(* Logix 5000 project; controller DUNEW2PLC1 vendor 1 type 14 code 221 rev 33.11; software revision 33.00; part 5 of 7 *)
(* tags used below, declared in another part *)
   AbortQueue : BOOL;
   ALL_EOT_GOOD : BOOL;
   btm_support_collision_ymax : DINT;
   btm_support_collision_ymin : DINT;
   ERROR_CODE : DINT;
   FRAME_LOC_FT_BTM : BOOL;
   FRAME_LOC_FT_MID : BOOL;
   FRAME_LOC_FT_TOP : BOOL;
   FRAME_LOC_HD_BTM : BOOL;
   FRAME_LOC_HD_MID : BOOL;
   FRAME_LOC_HD_TOP : BOOL;
   INIT_DONE : BOOL;
   mid_support_collision_ymax : DINT;
   mid_support_collision_ymin : DINT;
   MINUS_X_EOT : BOOL;
   MINUS_Y_EOT : BOOL;
   MOVE_TYPE : INT;   // 0 = No Move 1 = XY JOG 2 = XY Plane Move 3 = Z JOG 4 = Z Axis Move 5 = Toggle Latch Actuator 6 = Home the Latch Actuator
   NEXTSTATE : DINT;
   PLUS_X_EOT : BOOL;
   PLUS_Y_EOT : BOOL;
   STATE : DINT;   // CURRENT State Machine State
   STATE_REQUEST : DINT;
   top_support_collision_ymax : DINT;
   top_support_collision_ymin : DINT;
   X_axis : AXIS_CIP_DRIVE;
   X_XFER_OK : BOOL;   // If at the head, check head support arms. Same for foot
   X_Y : COORDINATE_SYSTEM;
   xz : COORDINATE_SYSTEM;
   xz_position_target : REAL[2];
   xz_speed : DINT;
   Y_axis : AXIS_CIP_DRIVE;
   Y_XFER_OK : BOOL;
   yz : COORDINATE_SYSTEM;
   yz_position_target : REAL[2];
   yz_speed : DINT;
   Z_axis : AXIS_CIP_DRIVE;
   Z_EOT : BOOL;
   Z_RETRACTED : BOOL;

PROGRAM state_10_error   (* main routine main *)
VAR
   error_axes_stopped_ob : BOOL;
   error_axes_stopped_sb : BOOL := 1;
   error_entry_ob : BOOL;
   error_entry_sb : BOOL;
   error_servo_off : BOOL;
   error_servoed_off_ob : BOOL;
   error_servoed_off_sb : BOOL;
   STATE10_IND : BOOL; {access Read Only}
   x_axis_mafr : MOTION_INSTRUCTION := (FLAGS := 33554432);
   x_axis_msf : MOTION_INSTRUCTION := (FLAGS := 33554432);
   xy_error_stop_control : MOTION_INSTRUCTION := (FLAGS := 704643072, DN := 1, PC := 1);
   y_axis_mafr : MOTION_INSTRUCTION := (FLAGS := 33554432);
   y_axis_msf : MOTION_INSTRUCTION := (FLAGS := 33554432);
   z_axis_error_stop_control : MOTION_INSTRUCTION := (FLAGS := 704643072, DN := 1, PC := 1);
   z_axis_mafr : MOTION_INSTRUCTION := (FLAGS := 33554432);
   z_axis_msf : MOTION_INSTRUCTION := (FLAGS := 33554432);
END_VAR

ROUTINE main   (* ladder *)
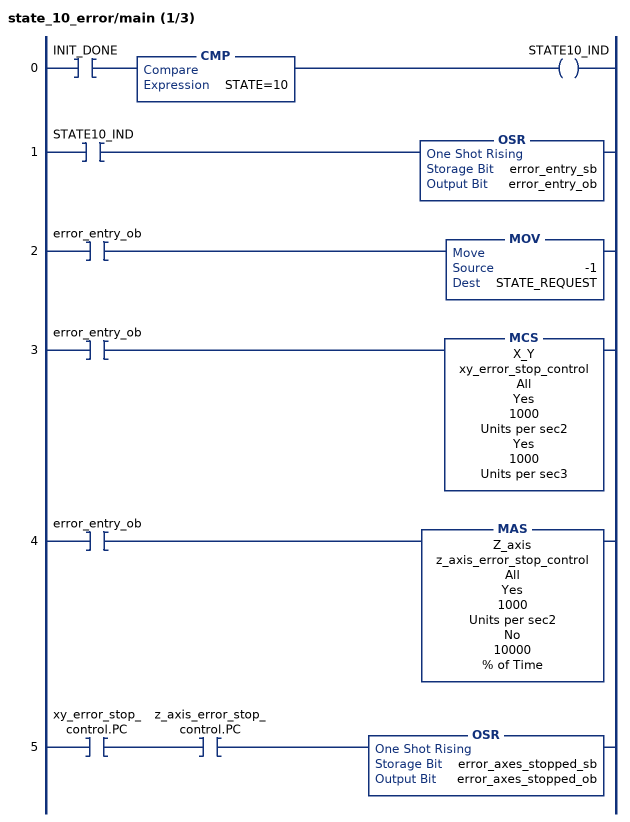
   0: XIC(INIT_DONE)CMP(STATE=10)OTE(STATE10_IND);
   1: XIC(STATE10_IND)OSR(error_entry_sb,error_entry_ob);
   2: XIC(error_entry_ob)MOV(-1,STATE_REQUEST);
   3: XIC(error_entry_ob)MCS(X_Y,xy_error_stop_control,All,Yes,1000,Units per sec2,Yes,1000,Units per sec3);
   4: XIC(error_entry_ob)MAS(Z_axis,z_axis_error_stop_control,All,Yes,1000,Units per sec2,No,10000,% of Time);
   5: XIC(xy_error_stop_control.PC)XIC(z_axis_error_stop_control.PC)OSR(error_axes_stopped_sb,error_axes_stopped_ob);
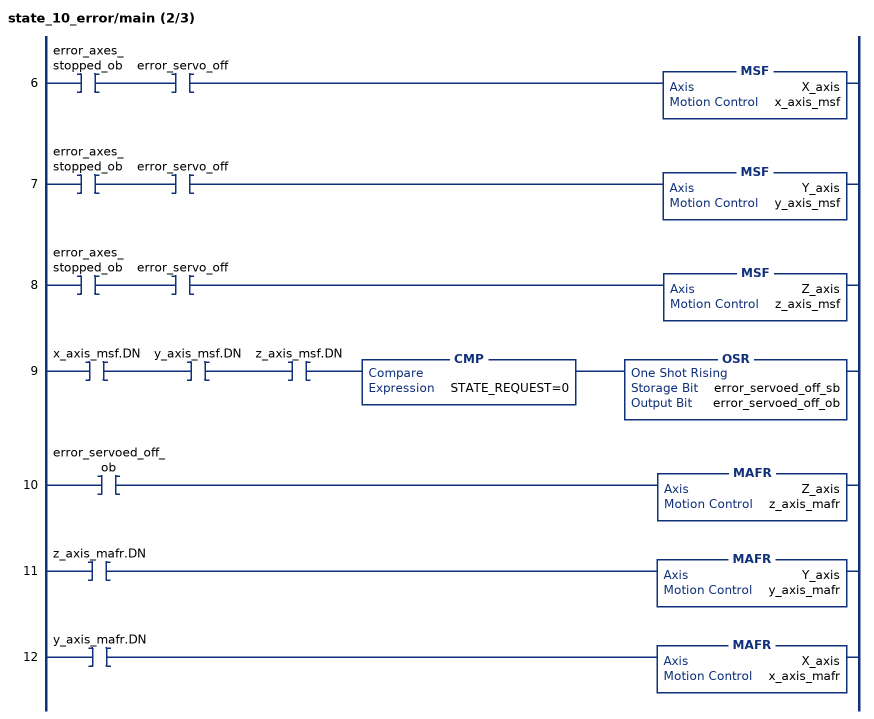
   6: XIC(error_axes_stopped_ob)XIC(error_servo_off)MSF(X_axis,x_axis_msf);
   7: XIC(error_axes_stopped_ob)XIC(error_servo_off)MSF(Y_axis,y_axis_msf);
   8: XIC(error_axes_stopped_ob)XIC(error_servo_off)MSF(Z_axis,z_axis_msf);
   9: XIC(x_axis_msf.DN)XIC(y_axis_msf.DN)XIC(z_axis_msf.DN)CMP(STATE_REQUEST=0)OSR(error_servoed_off_sb,error_servoed_off_ob);
   10: XIC(error_servoed_off_ob)MAFR(Z_axis,z_axis_mafr);
   11: XIC(z_axis_mafr.DN)MAFR(Y_axis,y_axis_mafr);
   12: XIC(y_axis_mafr.DN)MAFR(X_axis,x_axis_mafr);
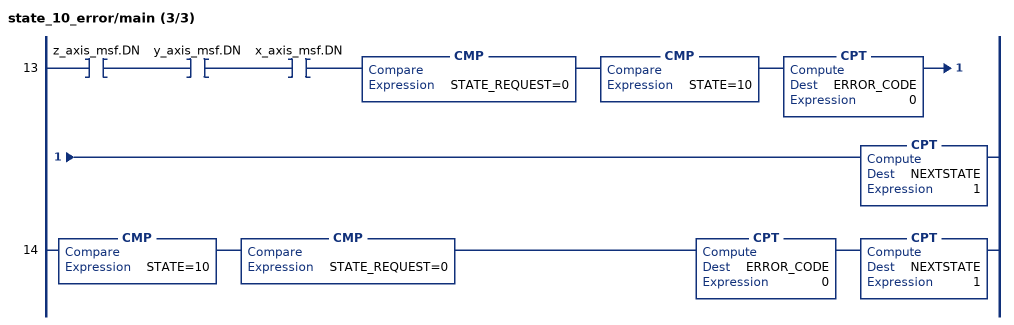
   13: XIC(z_axis_msf.DN)XIC(y_axis_msf.DN)XIC(x_axis_msf.DN)CMP(STATE_REQUEST=0)CMP(STATE=10)CPT(ERROR_CODE,0)CPT(NEXTSTATE,1);
   14: CMP(STATE=10)CMP(STATE_REQUEST=0)CPT(ERROR_CODE,0)CPT(NEXTSTATE,1);
END_ROUTINE
END_PROGRAM

PROGRAM state_11_eot_trip   (* main routine main *)
VAR
   eot_axes_enabled : BOOL := 1;
   eot_entry_ob : BOOL;
   eot_entry_sb : BOOL;
   eot_manual_ob : BOOL;
   eot_manual_sb : BOOL;
   eot_mso_start_ob : BOOL;
   eot_mso_start_sb : BOOL;
   eot_mso_x : MOTION_INSTRUCTION := (FLAGS := 536870912, DN := 1);
   eot_mso_y : MOTION_INSTRUCTION := (FLAGS := 536870912, DN := 1);
   eot_mso_z : MOTION_INSTRUCTION := (FLAGS := 536870912, DN := 1);
   eot_recover_ready : BOOL;
   eot_recovery_done : BOOL;
   eot_stop_x : MOTION_INSTRUCTION := (FLAGS := 671088640, DN := 1, PC := 1);
   eot_stop_xy : MOTION_INSTRUCTION := (FLAGS := 671088640, DN := 1, PC := 1);
   eot_stop_xz : MOTION_INSTRUCTION := (FLAGS := 671088640, DN := 1, PC := 1);
   eot_stop_y : MOTION_INSTRUCTION := (FLAGS := 671088640, DN := 1, PC := 1);
   eot_stop_yz : MOTION_INSTRUCTION := (FLAGS := 704643072, DN := 1, PC := 1);
   eot_stop_z : MOTION_INSTRUCTION := (FLAGS := 671088640, DN := 1, PC := 1);
   eot_stops_done : BOOL;
   STATE11_IND : BOOL; {access Read Only}
   x_minus_clear_ob : BOOL;
   x_minus_clear_sb : BOOL;
   x_minus_cleared : BOOL;
   x_minus_jog_active : BOOL;
   x_minus_jog_cmd : MOTION_INSTRUCTION;
   x_minus_jog_start_ob : BOOL;
   x_minus_jog_start_sb : BOOL;
   x_minus_jog_stop : MOTION_INSTRUCTION;
   x_minus_jog_timer : TIMER := (PRE := 10000);
   x_minus_mrp_cmd : MOTION_INSTRUCTION;
   x_minus_mrp_start_ob : BOOL;
   x_minus_mrp_start_sb : BOOL;
   x_minus_stop_req : BOOL;
   x_minus_timeout : BOOL;
   x_minus_trip : BOOL;
   x_plus_clear_ob : BOOL;
   x_plus_clear_sb : BOOL;
   x_plus_jog_active : BOOL;
   x_plus_jog_cmd : MOTION_INSTRUCTION := (FLAGS := 536870912, DN := 1);
   x_plus_jog_start_ob : BOOL;
   x_plus_jog_start_sb : BOOL;
   x_plus_jog_stop : MOTION_INSTRUCTION := (FLAGS := 671088640, DN := 1, PC := 1);
   x_plus_jog_timer : TIMER := (PRE := 10000);
   x_plus_stop_req : BOOL;
   x_plus_timeout : BOOL;
   x_plus_trip : BOOL;
   y_minus_clear_ob : BOOL;
   y_minus_clear_sb : BOOL;
   y_minus_cleared : BOOL;
   y_minus_jog_active : BOOL;
   y_minus_jog_cmd : MOTION_INSTRUCTION;
   y_minus_jog_start_ob : BOOL;
   y_minus_jog_start_sb : BOOL;
   y_minus_jog_stop : MOTION_INSTRUCTION;
   y_minus_jog_timer : TIMER := (PRE := 10000);
   y_minus_mrp_cmd : MOTION_INSTRUCTION;
   y_minus_mrp_start_ob : BOOL;
   y_minus_mrp_start_sb : BOOL;
   y_minus_stop_req : BOOL;
   y_minus_timeout : BOOL;
   y_minus_trip : BOOL;
   y_plus_clear_ob : BOOL;
   y_plus_clear_sb : BOOL;
   y_plus_jog_active : BOOL;
   y_plus_jog_cmd : MOTION_INSTRUCTION;
   y_plus_jog_start_ob : BOOL;
   y_plus_jog_start_sb : BOOL;
   y_plus_jog_stop : MOTION_INSTRUCTION;
   y_plus_jog_timer : TIMER := (PRE := 10000);
   y_plus_stop_req : BOOL;
   y_plus_timeout : BOOL;
   y_plus_trip : BOOL;
   z_recover_started : BOOL;
   z_trip : BOOL;
   z_zero_cmd : MOTION_INSTRUCTION;
   z_zero_start_ob : BOOL;
   z_zero_start_sb : BOOL;
END_VAR

ROUTINE main   (* ladder *)
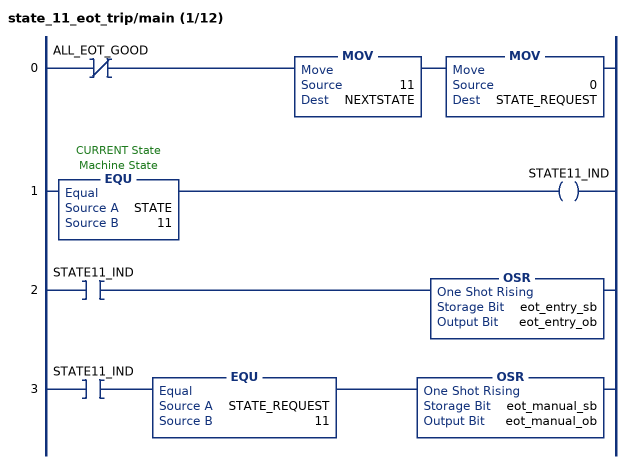
   0: XIO(ALL_EOT_GOOD)MOV(11,NEXTSTATE)MOV(0,STATE_REQUEST);
   1: EQU(STATE,11)OTE(STATE11_IND);
   2: XIC(STATE11_IND)OSR(eot_entry_sb,eot_entry_ob);
   3: XIC(STATE11_IND)EQU(STATE_REQUEST,11)OSR(eot_manual_sb,eot_manual_ob);
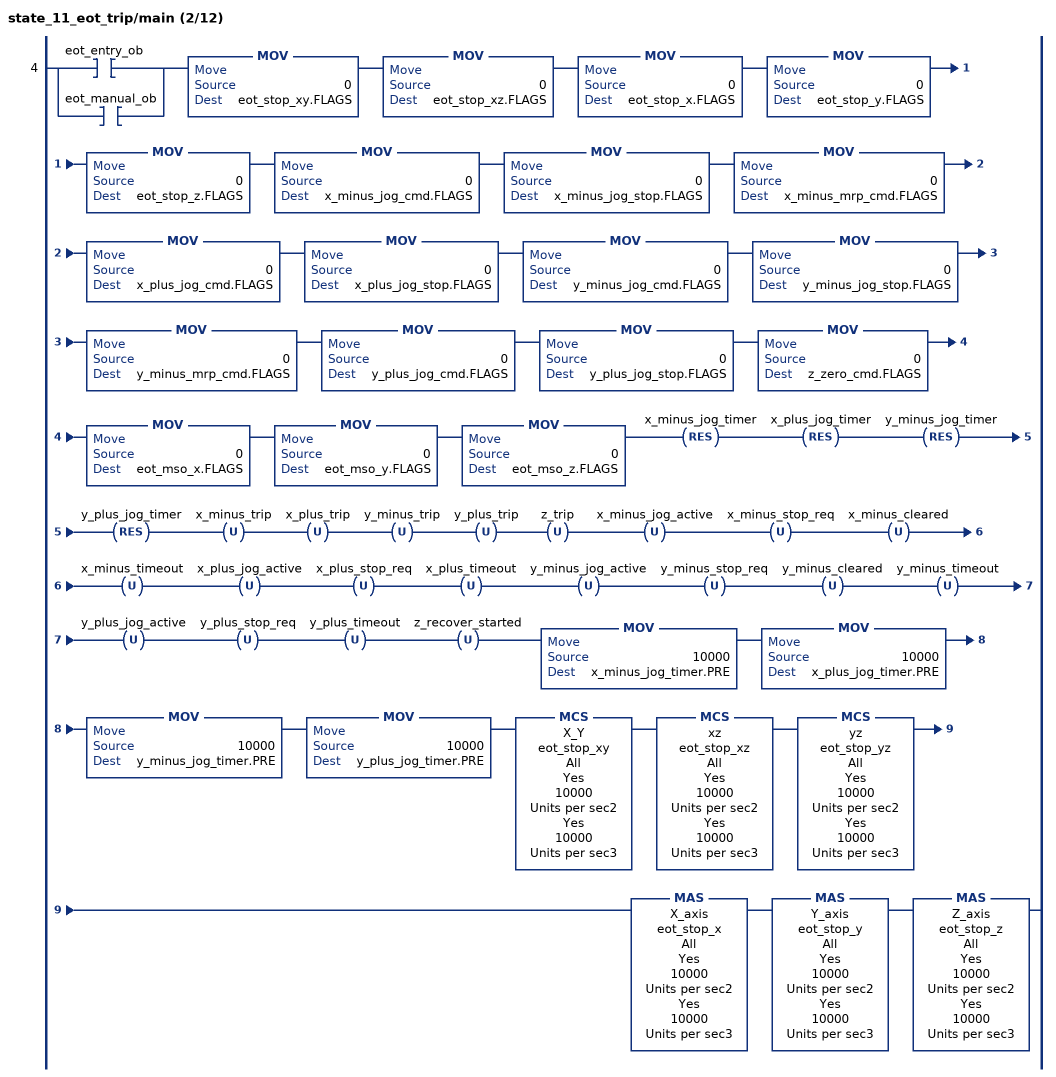
   4: [XIC(eot_entry_ob) ,XIC(eot_manual_ob) ]MOV(0,eot_stop_xy.FLAGS)MOV(0,eot_stop_xz.FLAGS)MOV(0,eot_stop_x.FLAGS)MOV(0,eot_stop_y.FLAGS)MOV(0,eot_stop_z.FLAGS)MOV(0,x_minus_jog_cmd.FLAGS)MOV(0,x_minus_jog_stop.FLAGS)MOV(0,x_minus_mrp_cmd.FLAGS)MOV(0,x_plus_jog_cmd.FLAGS)MOV(0,x_plus_jog_stop.FLAGS)MOV(0,y_minus_jog_cmd.FLAGS)MOV(0,y_minus_jog_stop.FLAGS)MOV(0,y_minus_mrp_cmd.FLAGS)MOV(0,y_plus_jog_cmd.FLAGS)MOV(0,y_plus_jog_stop.FLAGS)MOV(0,z_zero_cmd.FLAGS)MOV(0,eot_mso_x.FLAGS)MOV(0,eot_mso_y.FLAGS)MOV(0,eot_mso_z.FLAGS)RES(x_minus_jog_timer)RES(x_plus_jog_timer)RES(y_minus_jog_timer)RES(y_plus_jog_timer)OTU(x_minus_trip)OTU(x_plus_trip)OTU(y_minus_trip)OTU(y_plus_trip)OTU(z_trip)OTU(x_minus_jog_active)OTU(x_minus_stop_req)OTU(x_minus_cleared)OTU(x_minus_timeout)OTU(x_plus_jog_active)OTU(x_plus_stop_req)OTU(x_plus_timeout)OTU(y_minus_jog_active)OTU(y_minus_stop_req)OTU(y_minus_cleared)OTU(y_minus_timeout)OTU(y_plus_jog_active)OTU(y_plus_stop_req)OTU(y_plus_timeout)OTU(z_recover_started)MOV(10000,x_minus_jog_timer.PRE)MOV(10000,x_plus_jog_timer.PRE)MOV(10000,y_minus_jog_timer.PRE)MOV(10000,y_plus_jog_timer.PRE)MCS(X_Y,eot_stop_xy,All,Yes,10000,Units per sec2,Yes,10000,Units per sec3)MCS(xz,eot_stop_xz,All,Yes,10000,Units per sec2,Yes,10000,Units per sec3)MCS(yz,eot_stop_yz,All,Yes,10000,Units per sec2,Yes,10000,Units per sec3)MAS(X_axis,eot_stop_x,All,Yes,10000,Units per sec2,Yes,10000,Units per sec3)MAS(Y_axis,eot_stop_y,All,Yes,10000,Units per sec2,Yes,10000,Units per sec3)MAS(Z_axis,eot_stop_z,All,Yes,10000,Units per sec2,Yes,10000,Units per sec3);
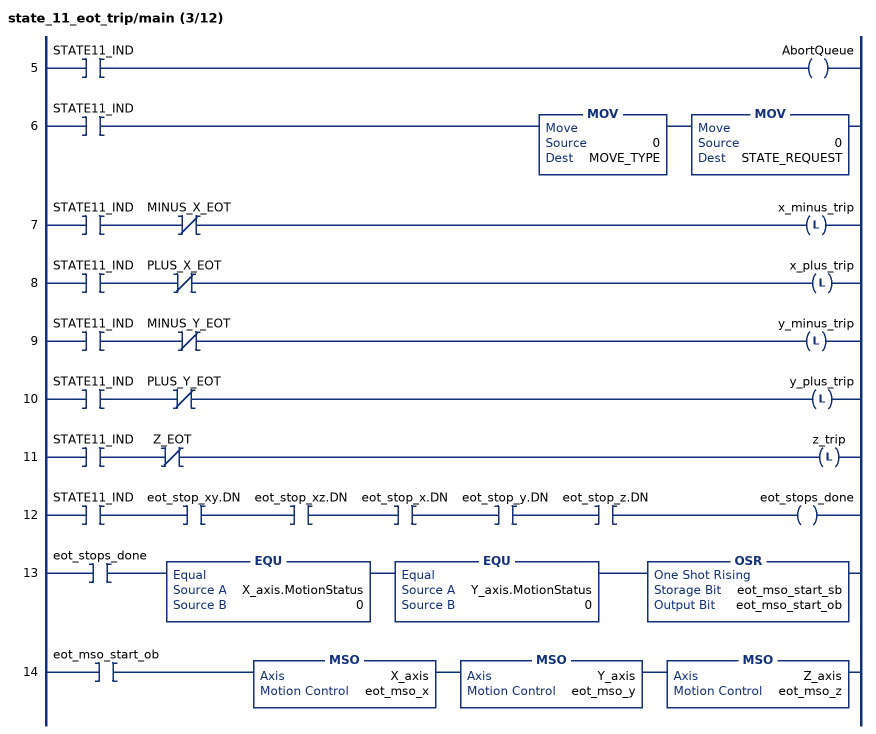
   5: XIC(STATE11_IND)OTE(AbortQueue);
   6: XIC(STATE11_IND)MOV(0,MOVE_TYPE)MOV(0,STATE_REQUEST);
   7: XIC(STATE11_IND)XIO(MINUS_X_EOT)OTL(x_minus_trip);
   8: XIC(STATE11_IND)XIO(PLUS_X_EOT)OTL(x_plus_trip);
   9: XIC(STATE11_IND)XIO(MINUS_Y_EOT)OTL(y_minus_trip);
   10: XIC(STATE11_IND)XIO(PLUS_Y_EOT)OTL(y_plus_trip);
   11: XIC(STATE11_IND)XIO(Z_EOT)OTL(z_trip);
   12: XIC(STATE11_IND)XIC(eot_stop_xy.DN)XIC(eot_stop_xz.DN)XIC(eot_stop_x.DN)XIC(eot_stop_y.DN)XIC(eot_stop_z.DN)OTE(eot_stops_done);
   13: XIC(eot_stops_done)EQU(X_axis.MotionStatus,0)EQU(Y_axis.MotionStatus,0)OSR(eot_mso_start_sb,eot_mso_start_ob);
   14: XIC(eot_mso_start_ob)MSO(X_axis,eot_mso_x)MSO(Y_axis,eot_mso_y)MSO(Z_axis,eot_mso_z);
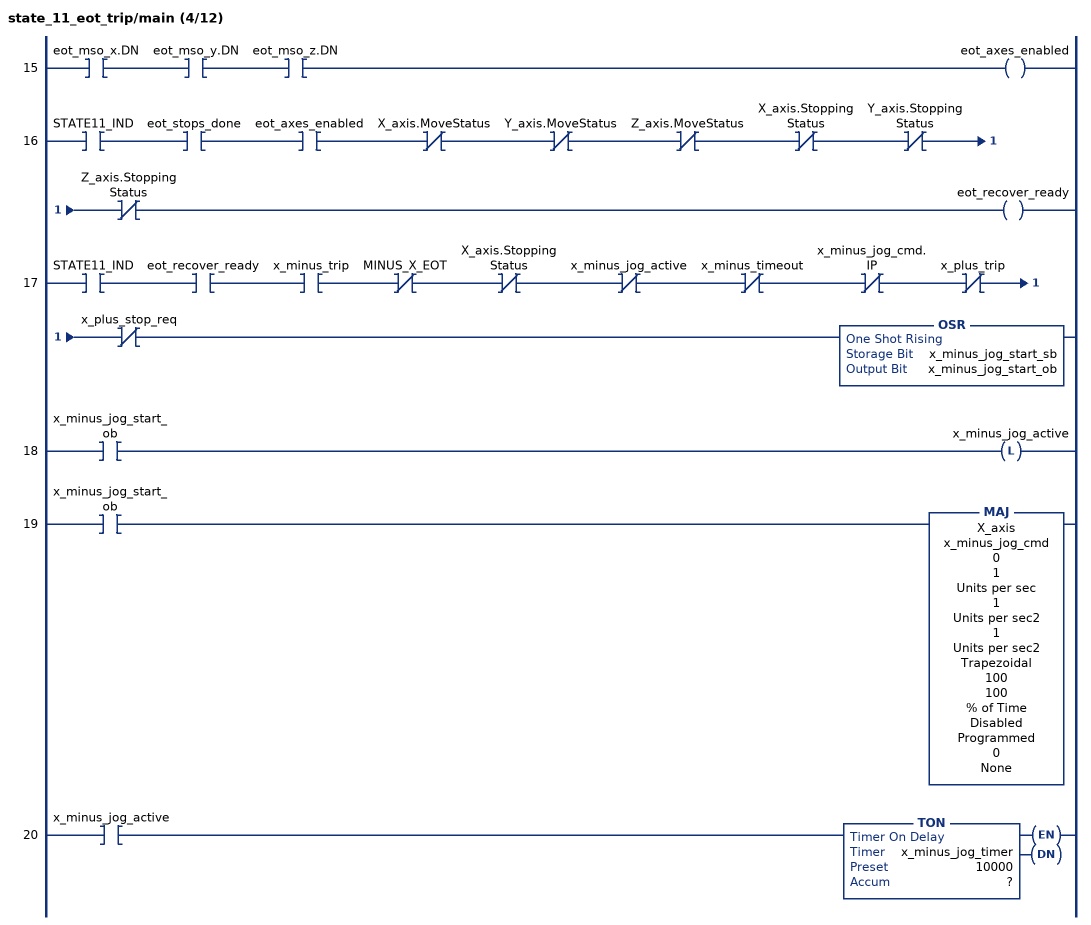
   15: XIC(eot_mso_x.DN)XIC(eot_mso_y.DN)XIC(eot_mso_z.DN)OTE(eot_axes_enabled);
   16: XIC(STATE11_IND)XIC(eot_stops_done)XIC(eot_axes_enabled)XIO(X_axis.MoveStatus)XIO(Y_axis.MoveStatus)XIO(Z_axis.MoveStatus)XIO(X_axis.StoppingStatus)XIO(Y_axis.StoppingStatus)XIO(Z_axis.StoppingStatus)OTE(eot_recover_ready);
   17: XIC(STATE11_IND)XIC(eot_recover_ready)XIC(x_minus_trip)XIO(MINUS_X_EOT)XIO(X_axis.StoppingStatus)XIO(x_minus_jog_active)XIO(x_minus_timeout)XIO(x_minus_jog_cmd.IP)XIO(x_plus_trip)XIO(x_plus_stop_req)OSR(x_minus_jog_start_sb,x_minus_jog_start_ob);
   18: XIC(x_minus_jog_start_ob)OTL(x_minus_jog_active);
   19: XIC(x_minus_jog_start_ob)MAJ(X_axis,x_minus_jog_cmd,0,1,Units per sec,1,Units per sec2,1,Units per sec2,Trapezoidal,100,100,% of Time,Disabled,Programmed,0,None);
   20: XIC(x_minus_jog_active)TON(x_minus_jog_timer,?,?);
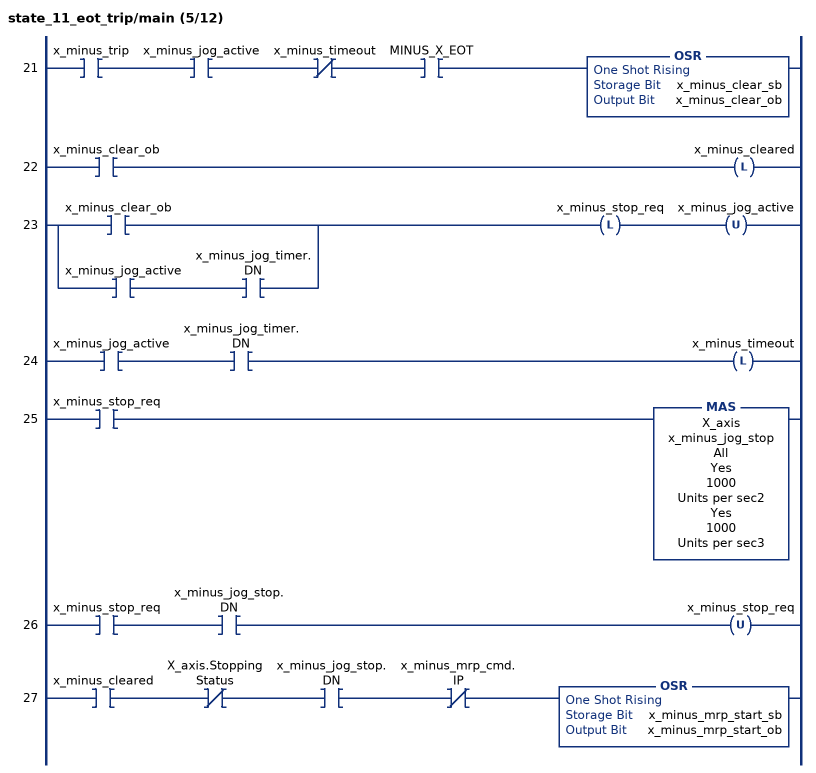
   21: XIC(x_minus_trip)XIC(x_minus_jog_active)XIO(x_minus_timeout)XIC(MINUS_X_EOT)OSR(x_minus_clear_sb,x_minus_clear_ob);
   22: XIC(x_minus_clear_ob)OTL(x_minus_cleared);
   23: [XIC(x_minus_clear_ob) ,XIC(x_minus_jog_active) XIC(x_minus_jog_timer.DN) ]OTL(x_minus_stop_req)OTU(x_minus_jog_active);
   24: XIC(x_minus_jog_active)XIC(x_minus_jog_timer.DN)OTL(x_minus_timeout);
   25: XIC(x_minus_stop_req)MAS(X_axis,x_minus_jog_stop,All,Yes,1000,Units per sec2,Yes,1000,Units per sec3);
   26: XIC(x_minus_stop_req)XIC(x_minus_jog_stop.DN)OTU(x_minus_stop_req);
   27: XIC(x_minus_cleared)XIO(X_axis.StoppingStatus)XIC(x_minus_jog_stop.DN)XIO(x_minus_mrp_cmd.IP)OSR(x_minus_mrp_start_sb,x_minus_mrp_start_ob);
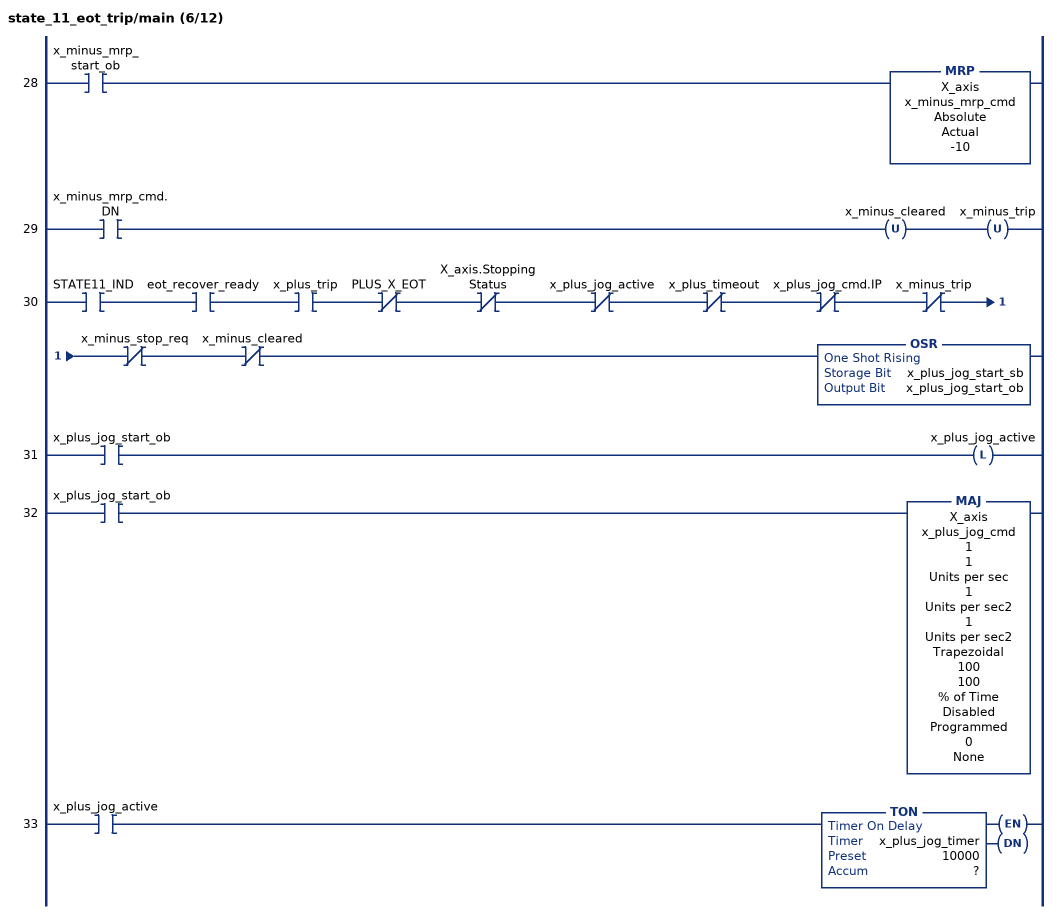
   28: XIC(x_minus_mrp_start_ob)MRP(X_axis,x_minus_mrp_cmd,Absolute,Actual,-10);
   29: XIC(x_minus_mrp_cmd.DN)OTU(x_minus_cleared)OTU(x_minus_trip);
   30: XIC(STATE11_IND)XIC(eot_recover_ready)XIC(x_plus_trip)XIO(PLUS_X_EOT)XIO(X_axis.StoppingStatus)XIO(x_plus_jog_active)XIO(x_plus_timeout)XIO(x_plus_jog_cmd.IP)XIO(x_minus_trip)XIO(x_minus_stop_req)XIO(x_minus_cleared)OSR(x_plus_jog_start_sb,x_plus_jog_start_ob);
   31: XIC(x_plus_jog_start_ob)OTL(x_plus_jog_active);
   32: XIC(x_plus_jog_start_ob)MAJ(X_axis,x_plus_jog_cmd,1,1,Units per sec,1,Units per sec2,1,Units per sec2,Trapezoidal,100,100,% of Time,Disabled,Programmed,0,None);
   33: XIC(x_plus_jog_active)TON(x_plus_jog_timer,?,?);
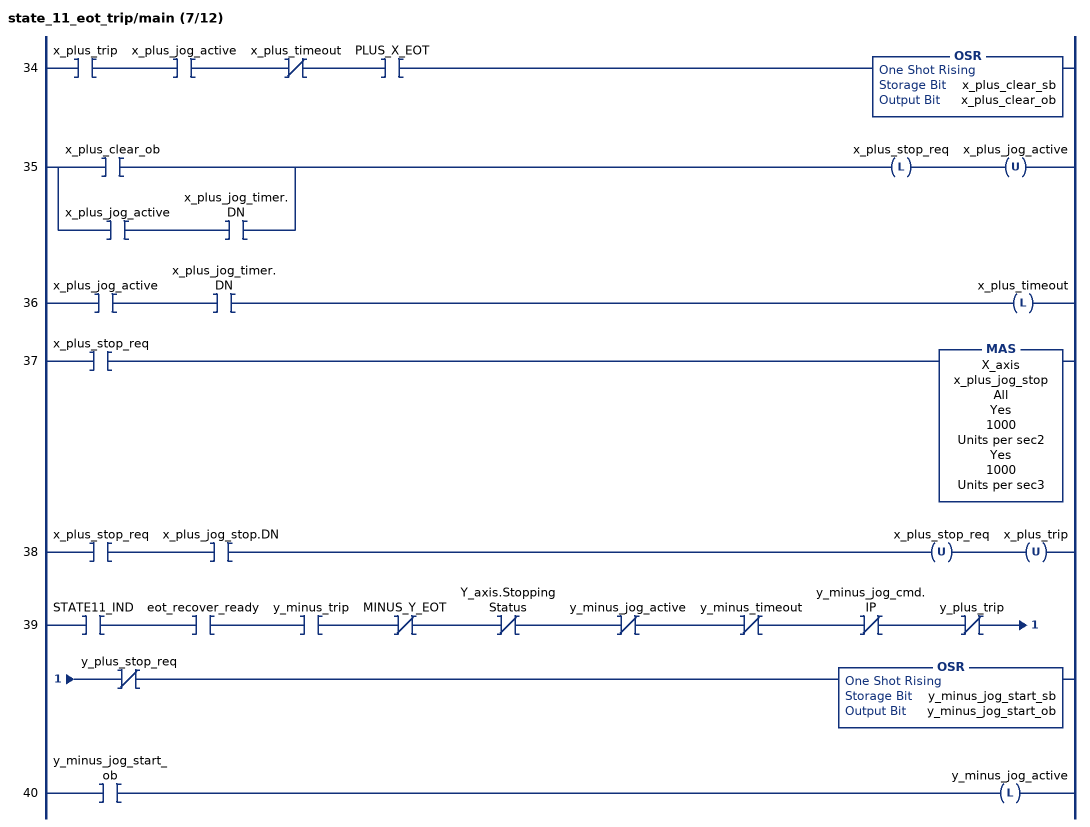
   34: XIC(x_plus_trip)XIC(x_plus_jog_active)XIO(x_plus_timeout)XIC(PLUS_X_EOT)OSR(x_plus_clear_sb,x_plus_clear_ob);
   35: [XIC(x_plus_clear_ob) ,XIC(x_plus_jog_active) XIC(x_plus_jog_timer.DN) ]OTL(x_plus_stop_req)OTU(x_plus_jog_active);
   36: XIC(x_plus_jog_active)XIC(x_plus_jog_timer.DN)OTL(x_plus_timeout);
   37: XIC(x_plus_stop_req)MAS(X_axis,x_plus_jog_stop,All,Yes,1000,Units per sec2,Yes,1000,Units per sec3);
   38: XIC(x_plus_stop_req)XIC(x_plus_jog_stop.DN)OTU(x_plus_stop_req)OTU(x_plus_trip);
   39: XIC(STATE11_IND)XIC(eot_recover_ready)XIC(y_minus_trip)XIO(MINUS_Y_EOT)XIO(Y_axis.StoppingStatus)XIO(y_minus_jog_active)XIO(y_minus_timeout)XIO(y_minus_jog_cmd.IP)XIO(y_plus_trip)XIO(y_plus_stop_req)OSR(y_minus_jog_start_sb,y_minus_jog_start_ob);
   40: XIC(y_minus_jog_start_ob)OTL(y_minus_jog_active);
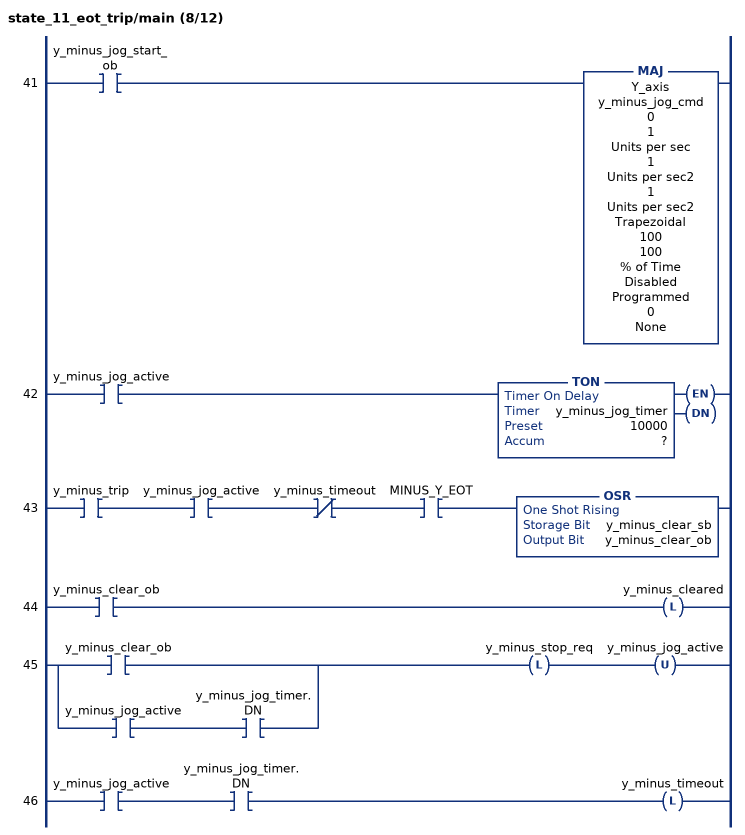
   41: XIC(y_minus_jog_start_ob)MAJ(Y_axis,y_minus_jog_cmd,0,1,Units per sec,1,Units per sec2,1,Units per sec2,Trapezoidal,100,100,% of Time,Disabled,Programmed,0,None);
   42: XIC(y_minus_jog_active)TON(y_minus_jog_timer,?,?);
   43: XIC(y_minus_trip)XIC(y_minus_jog_active)XIO(y_minus_timeout)XIC(MINUS_Y_EOT)OSR(y_minus_clear_sb,y_minus_clear_ob);
   44: XIC(y_minus_clear_ob)OTL(y_minus_cleared);
   45: [XIC(y_minus_clear_ob) ,XIC(y_minus_jog_active) XIC(y_minus_jog_timer.DN) ]OTL(y_minus_stop_req)OTU(y_minus_jog_active);
   46: XIC(y_minus_jog_active)XIC(y_minus_jog_timer.DN)OTL(y_minus_timeout);
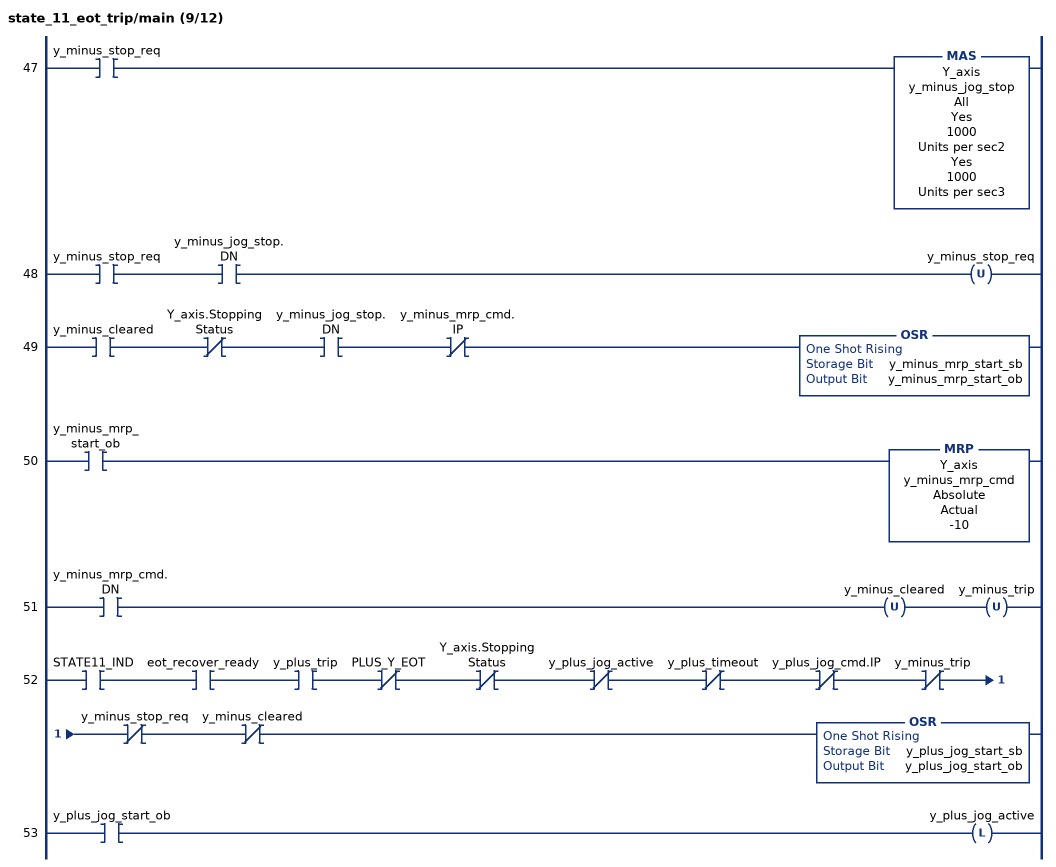
   47: XIC(y_minus_stop_req)MAS(Y_axis,y_minus_jog_stop,All,Yes,1000,Units per sec2,Yes,1000,Units per sec3);
   48: XIC(y_minus_stop_req)XIC(y_minus_jog_stop.DN)OTU(y_minus_stop_req);
   49: XIC(y_minus_cleared)XIO(Y_axis.StoppingStatus)XIC(y_minus_jog_stop.DN)XIO(y_minus_mrp_cmd.IP)OSR(y_minus_mrp_start_sb,y_minus_mrp_start_ob);
   50: XIC(y_minus_mrp_start_ob)MRP(Y_axis,y_minus_mrp_cmd,Absolute,Actual,-10);
   51: XIC(y_minus_mrp_cmd.DN)OTU(y_minus_cleared)OTU(y_minus_trip);
   52: XIC(STATE11_IND)XIC(eot_recover_ready)XIC(y_plus_trip)XIO(PLUS_Y_EOT)XIO(Y_axis.StoppingStatus)XIO(y_plus_jog_active)XIO(y_plus_timeout)XIO(y_plus_jog_cmd.IP)XIO(y_minus_trip)XIO(y_minus_stop_req)XIO(y_minus_cleared)OSR(y_plus_jog_start_sb,y_plus_jog_start_ob);
   53: XIC(y_plus_jog_start_ob)OTL(y_plus_jog_active);
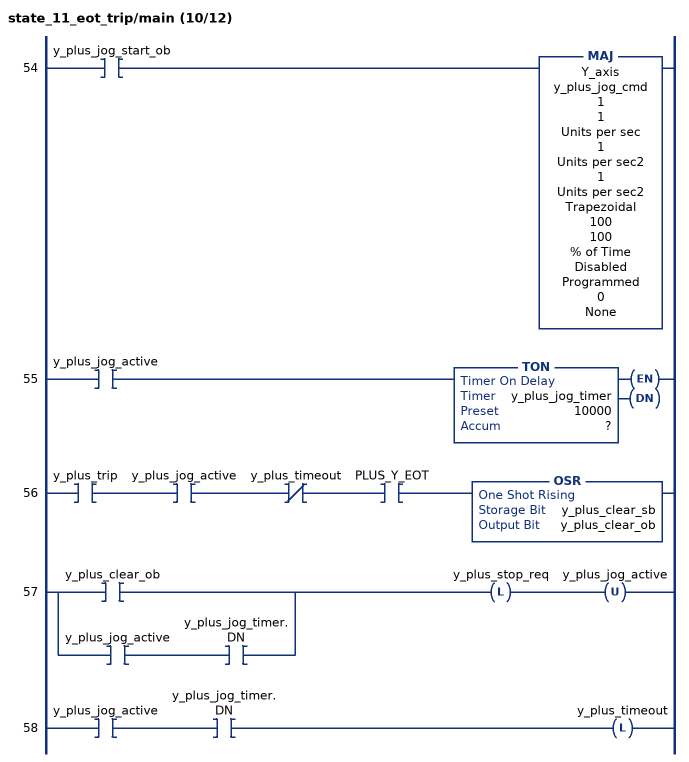
   54: XIC(y_plus_jog_start_ob)MAJ(Y_axis,y_plus_jog_cmd,1,1,Units per sec,1,Units per sec2,1,Units per sec2,Trapezoidal,100,100,% of Time,Disabled,Programmed,0,None);
   55: XIC(y_plus_jog_active)TON(y_plus_jog_timer,?,?);
   56: XIC(y_plus_trip)XIC(y_plus_jog_active)XIO(y_plus_timeout)XIC(PLUS_Y_EOT)OSR(y_plus_clear_sb,y_plus_clear_ob);
   57: [XIC(y_plus_clear_ob) ,XIC(y_plus_jog_active) XIC(y_plus_jog_timer.DN) ]OTL(y_plus_stop_req)OTU(y_plus_jog_active);
   58: XIC(y_plus_jog_active)XIC(y_plus_jog_timer.DN)OTL(y_plus_timeout);
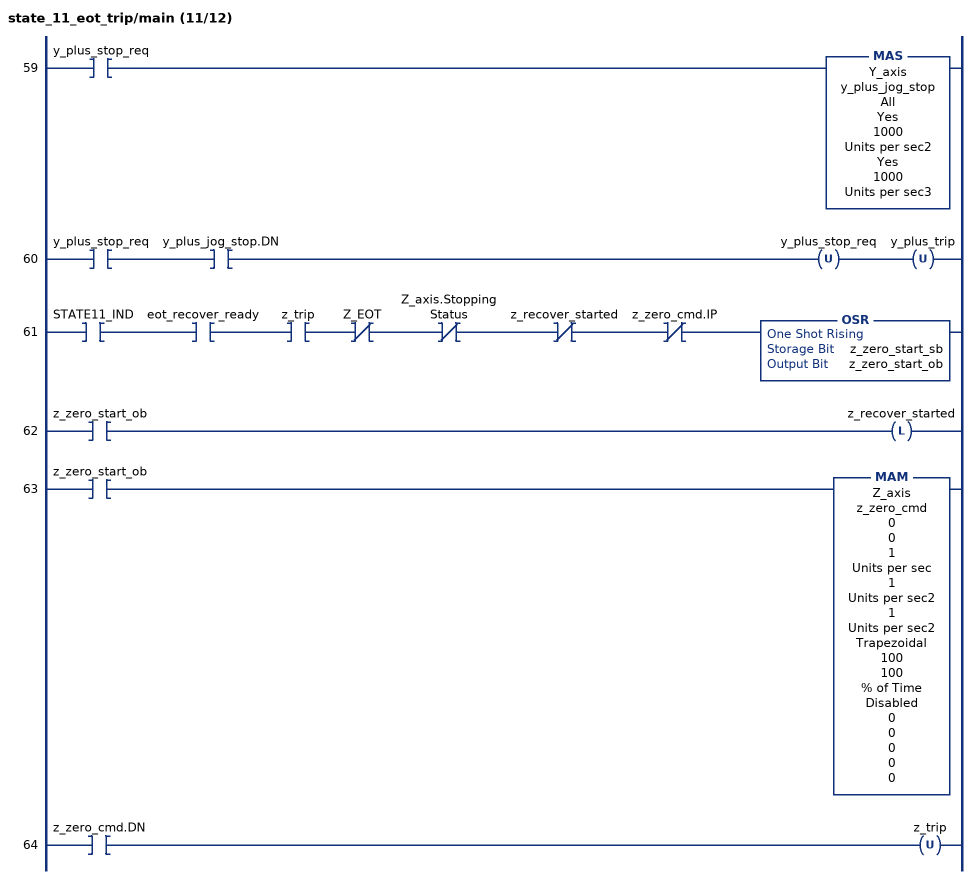
   59: XIC(y_plus_stop_req)MAS(Y_axis,y_plus_jog_stop,All,Yes,1000,Units per sec2,Yes,1000,Units per sec3);
   60: XIC(y_plus_stop_req)XIC(y_plus_jog_stop.DN)OTU(y_plus_stop_req)OTU(y_plus_trip);
   61: XIC(STATE11_IND)XIC(eot_recover_ready)XIC(z_trip)XIO(Z_EOT)XIO(Z_axis.StoppingStatus)XIO(z_recover_started)XIO(z_zero_cmd.IP)OSR(z_zero_start_sb,z_zero_start_ob);
   62: XIC(z_zero_start_ob)OTL(z_recover_started);
   63: XIC(z_zero_start_ob)MAM(Z_axis,z_zero_cmd,0,0,1,Units per sec,1,Units per sec2,1,Units per sec2,Trapezoidal,100,100,% of Time,Disabled,0,0,0,0,0);
   64: XIC(z_zero_cmd.DN)OTU(z_trip);
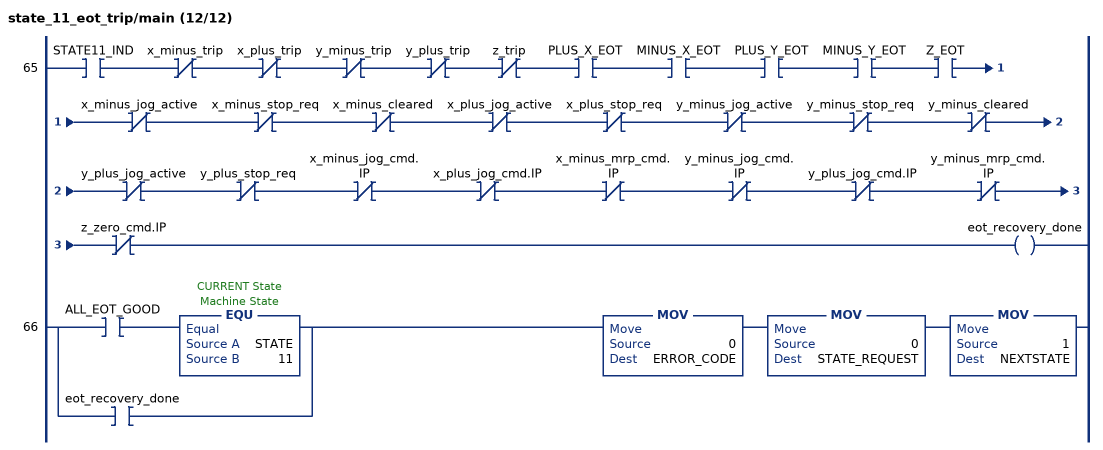
   65: XIC(STATE11_IND)XIO(x_minus_trip)XIO(x_plus_trip)XIO(y_minus_trip)XIO(y_plus_trip)XIO(z_trip)XIC(PLUS_X_EOT)XIC(MINUS_X_EOT)XIC(PLUS_Y_EOT)XIC(MINUS_Y_EOT)XIC(Z_EOT)XIO(x_minus_jog_active)XIO(x_minus_stop_req)XIO(x_minus_cleared)XIO(x_plus_jog_active)XIO(x_plus_stop_req)XIO(y_minus_jog_active)XIO(y_minus_stop_req)XIO(y_minus_cleared)XIO(y_plus_jog_active)XIO(y_plus_stop_req)XIO(x_minus_jog_cmd.IP)XIO(x_plus_jog_cmd.IP)XIO(x_minus_mrp_cmd.IP)XIO(y_minus_jog_cmd.IP)XIO(y_plus_jog_cmd.IP)XIO(y_minus_mrp_cmd.IP)XIO(z_zero_cmd.IP)OTE(eot_recovery_done);
   66: [XIC(ALL_EOT_GOOD) EQU(STATE,11) ,XIC(eot_recovery_done) ]MOV(0,ERROR_CODE)MOV(0,STATE_REQUEST)MOV(1,NEXTSTATE);
END_ROUTINE
END_PROGRAM

PROGRAM state_12_move_xz   (* main routine main *)
VAR
   STATE12_IND : BOOL;
   xy_stop : MOTION_INSTRUCTION := (FLAGS := 33554432);
   xz_main_move : MOTION_INSTRUCTION := (FLAGS := 33554432);
   xz_stop : MOTION_INSTRUCTION := (FLAGS := 33554432);
   y_axis_stop : MOTION_INSTRUCTION := (FLAGS := 33554432);
END_VAR

ROUTINE main   (* ladder *)
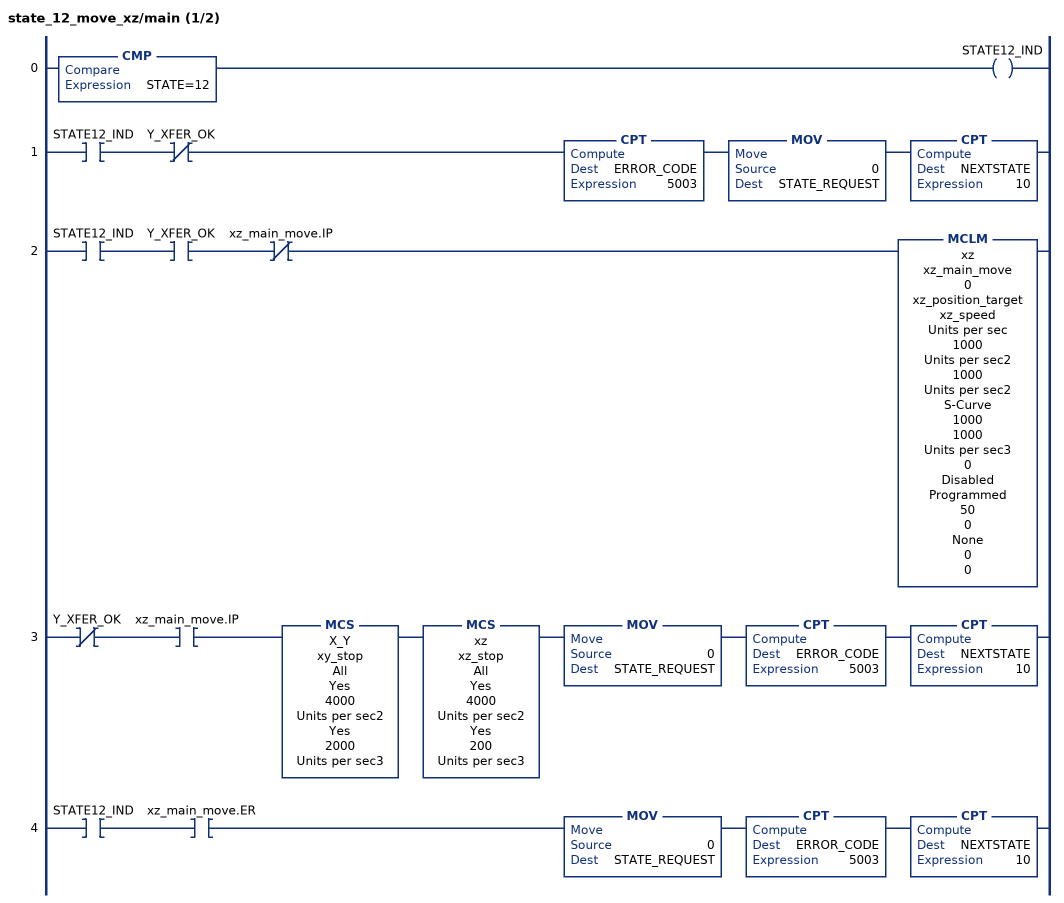
   0: CMP(STATE=12)OTE(STATE12_IND);
   1: XIC(STATE12_IND)XIO(Y_XFER_OK)CPT(ERROR_CODE,5003)MOV(0,STATE_REQUEST)CPT(NEXTSTATE,10);
   2: XIC(STATE12_IND)XIC(Y_XFER_OK)XIO(xz_main_move.IP)MCLM(xz,xz_main_move,0,xz_position_target,xz_speed,Units per sec,1000,Units per sec2,1000,Units per sec2,S-Curve,1000,1000,Units per sec3,0,Disabled,Programmed,50,0,None,0,0);
   3: XIO(Y_XFER_OK)XIC(xz_main_move.IP)MCS(X_Y,xy_stop,All,Yes,4000,Units per sec2,Yes,2000,Units per sec3)MCS(xz,xz_stop,All,Yes,4000,Units per sec2,Yes,200,Units per sec3)MOV(0,STATE_REQUEST)CPT(ERROR_CODE,5003)CPT(NEXTSTATE,10);
   4: XIC(STATE12_IND)XIC(xz_main_move.ER)MOV(0,STATE_REQUEST)CPT(ERROR_CODE,5003)CPT(NEXTSTATE,10);
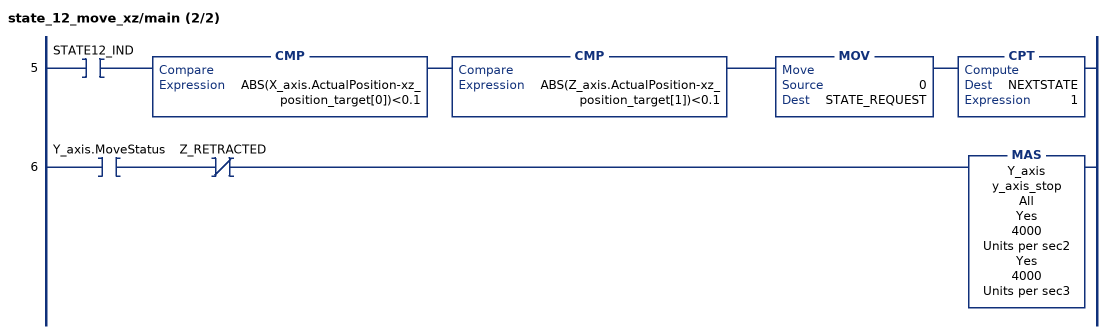
   5: XIC(STATE12_IND)CMP(ABS(X_axis.ActualPosition-xz_position_target[0])<0.1)CMP(ABS(Z_axis.ActualPosition-xz_position_target[1])<0.1)MOV(0,STATE_REQUEST)CPT(NEXTSTATE,1);
   6: XIC(Y_axis.MoveStatus)XIO(Z_RETRACTED)MAS(Y_axis,y_axis_stop,All,Yes,4000,Units per sec2,Yes,4000,Units per sec3);
END_ROUTINE
END_PROGRAM

PROGRAM state_13_move_yz   (* main routine main *)
VAR
   null : BOOL;
   oneshotob_yz_trigger : BOOL;
   oneshotsb_yz_trigger : BOOL;
   STATE13_IND : BOOL;
   state_13_entry_osr : BOOL;
   x_axis_stop : MOTION_INSTRUCTION := (FLAGS := 33554432);
   x_in_foot_transfer_zone : BOOL;
   x_in_head_transfer_zone : BOOL;
   xy_stop : MOTION_INSTRUCTION := (FLAGS := 33554432);
   yz_main_move : MOTION_INSTRUCTION := (FLAGS := 33554432);
   yz_stop : MOTION_INSTRUCTION := (FLAGS := 33554432);
   yz_target_collision_bttm : BOOL := 1;
   yz_target_collision_mid : BOOL;
   yz_target_collision_top : BOOL;
   yz_target_support_collision : BOOL;
END_VAR

ROUTINE main   (* ladder *)
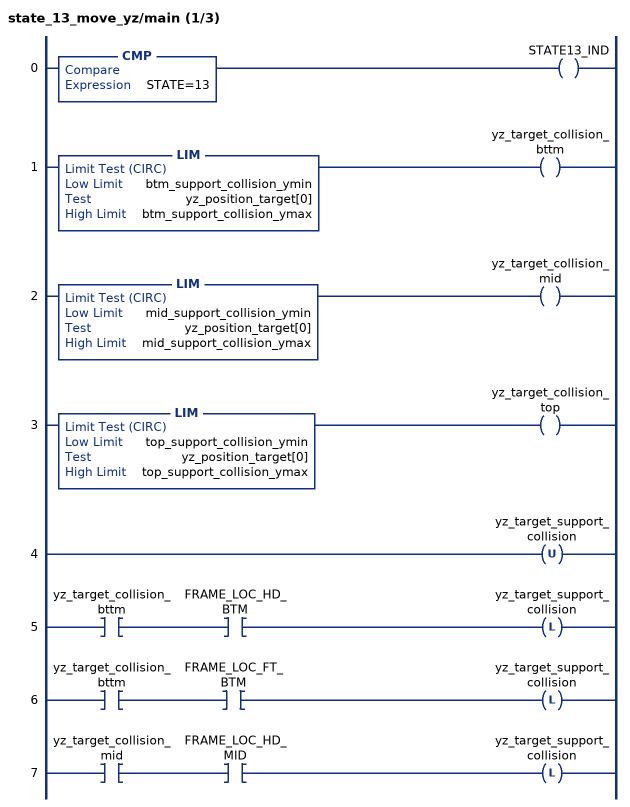
   0: CMP(STATE=13)OTE(STATE13_IND);
   1: LIM(btm_support_collision_ymin,yz_position_target[0],btm_support_collision_ymax)OTE(yz_target_collision_bttm);
   2: LIM(mid_support_collision_ymin,yz_position_target[0],mid_support_collision_ymax)OTE(yz_target_collision_mid);
   3: LIM(top_support_collision_ymin,yz_position_target[0],top_support_collision_ymax)OTE(yz_target_collision_top);
   4: OTU(yz_target_support_collision);
   5: XIC(yz_target_collision_bttm)XIC(FRAME_LOC_HD_BTM)OTL(yz_target_support_collision);
   6: XIC(yz_target_collision_bttm)XIC(FRAME_LOC_FT_BTM)OTL(yz_target_support_collision);
   7: XIC(yz_target_collision_mid)XIC(FRAME_LOC_HD_MID)OTL(yz_target_support_collision);
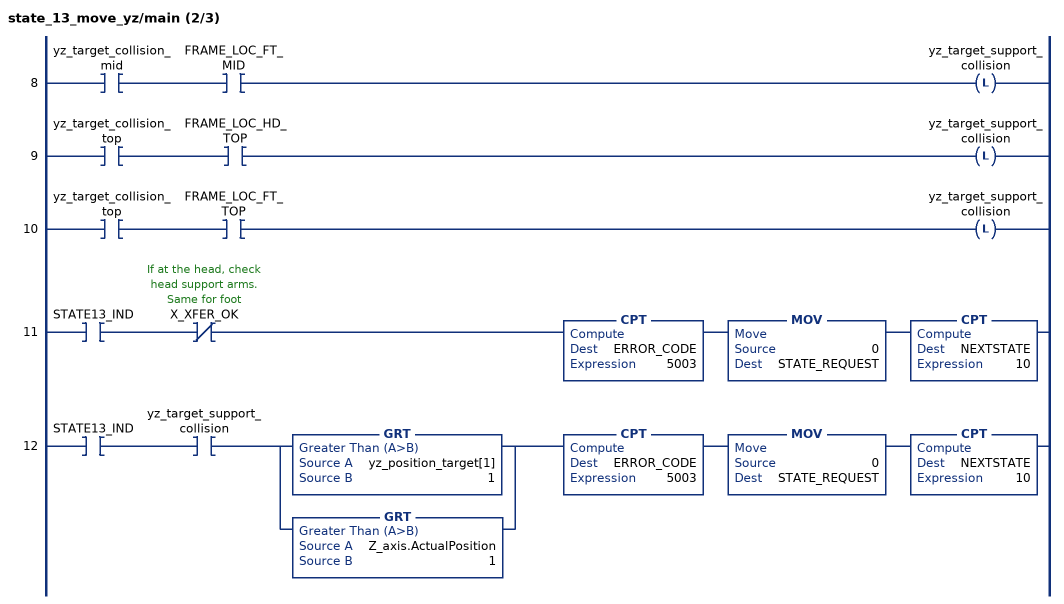
   8: XIC(yz_target_collision_mid)XIC(FRAME_LOC_FT_MID)OTL(yz_target_support_collision);
   9: XIC(yz_target_collision_top)XIC(FRAME_LOC_HD_TOP)OTL(yz_target_support_collision);
   10: XIC(yz_target_collision_top)XIC(FRAME_LOC_FT_TOP)OTL(yz_target_support_collision);
   11: XIC(STATE13_IND)XIO(X_XFER_OK)CPT(ERROR_CODE,5003)MOV(0,STATE_REQUEST)CPT(NEXTSTATE,10);
   12: XIC(STATE13_IND)XIC(yz_target_support_collision)[GRT(yz_position_target[1],1) ,GRT(Z_axis.ActualPosition,1) ]CPT(ERROR_CODE,5003)MOV(0,STATE_REQUEST)CPT(NEXTSTATE,10);
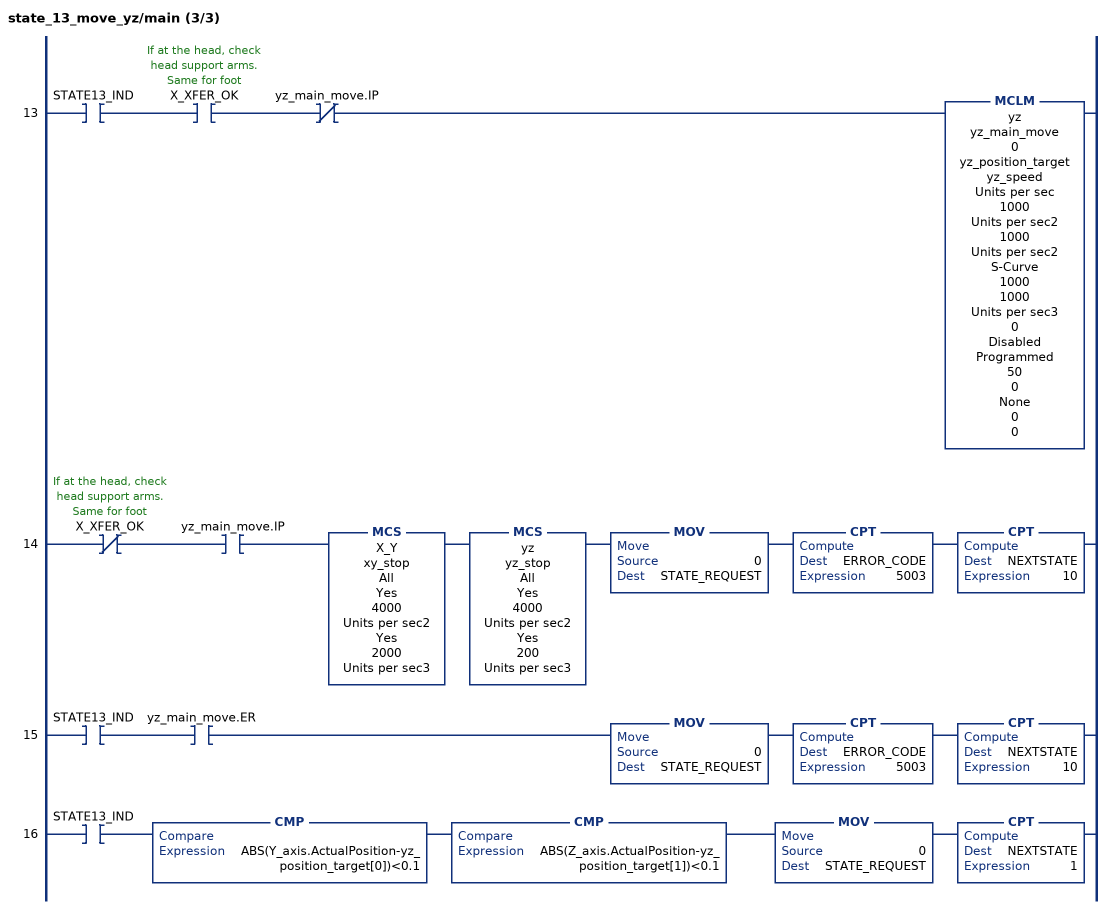
   13: XIC(STATE13_IND)XIC(X_XFER_OK)XIO(yz_main_move.IP)MCLM(yz,yz_main_move,0,yz_position_target,yz_speed,Units per sec,1000,Units per sec2,1000,Units per sec2,S-Curve,1000,1000,Units per sec3,0,Disabled,Programmed,50,0,None,0,0);
   14: XIO(X_XFER_OK)XIC(yz_main_move.IP)MCS(X_Y,xy_stop,All,Yes,4000,Units per sec2,Yes,2000,Units per sec3)MCS(yz,yz_stop,All,Yes,4000,Units per sec2,Yes,200,Units per sec3)MOV(0,STATE_REQUEST)CPT(ERROR_CODE,5003)CPT(NEXTSTATE,10);
   15: XIC(STATE13_IND)XIC(yz_main_move.ER)MOV(0,STATE_REQUEST)CPT(ERROR_CODE,5003)CPT(NEXTSTATE,10);
   16: XIC(STATE13_IND)CMP(ABS(Y_axis.ActualPosition-yz_position_target[0])<0.1)CMP(ABS(Z_axis.ActualPosition-yz_position_target[1])<0.1)MOV(0,STATE_REQUEST)CPT(NEXTSTATE,1);
END_ROUTINE
END_PROGRAM
